# EPICS substitutions: siteApps/EtherCat/m-epics-ecat2db/db/ecat2el2004.substitutions
file ecat2slave.template
{
	pattern {DEVICENAME}
		{EL2004}
}

file ecat2el20xxel2124DO.template
{
	pattern {CH_ID, PDO_IDX}
		{$(MOD_ID)-DO1, 0}
		{$(MOD_ID)-DO2, 1}
		{$(MOD_ID)-DO3, 2}
		{$(MOD_ID)-DO4, 3}
}
